TYPE DW_TO_REAL :
UNION
	IntAsWord : ARRAY[0..1] OF WORD;
	IntAsReal: REAL;
END_UNION
END_TYPE

(* stored: Version 1.1.0.1, ProductVersion 3.1.0.26
   DUT DW_TO_REAL: Id {ff45140b-45d5-402d-b726-1e45be2f2921} *)
